Staubli VAL3: CartesianVel.pjx

Parameters version=s7.9.1 stackSize=5000 millimeterUnit=true
Data file=CartesianVel.dtx
